// TwinCAT 3 PLC project TcoElements
// Title: TcoElements
// Company: Vortex.Library
// ProjectVersion: 0.6.0.913
// ProgramVersion: 3.1.4024.12
// libraries:
//   Tc2_Standard, * (Beckhoff Automation GmbH)
//   Tc2_System, * (Beckhoff Automation GmbH)
//   Tc3_Module, * (Beckhoff Automation GmbH)
//   TcoCore, 0.6.0.913 (Vortex.Library)
//   TcoUtilities, 0.6.0.913 (Vortex.Library)
// project tree:
//   Analog/TcoAi/ TcoAiAny.TcPOU, TcoAi.TcPOU, TcoAiConfig.TcDUT, TcoAiStatus.TcDUT
//   Analog/TcoAo/ TcoAoConfig.TcDUT, TcoAoStatus.TcDUT, TcoAo.TcPOU
//   Carousel/Base/ TcoCarouselBase.TcPOU
//   Carousel/Structs/ eTcoCarouselDirection.TcDUT, TcoCarouselConfig.TcDUT, TcoCarouselStatus.TcDUT
//   Carousel/Tasks/ TcoTurnTableTask.TcPOU
//   Carousel/ TcoCarousel.TcPOU
//   Digital/TcoDi/ TcoDi.TcPOU, TcoDiConfig.TcDUT
//   Digital/TcoDo/ TcoDo.TcPOU
//   / PlcTask.TcTTO
//   POUs/ MAIN.TcPOU
// real-time tasks:
//   TASK PlcTask: cycle T#10ms, priority 20, ADS port 350
//   TASK PlcTask1: cycle T#10ms, priority 21, ADS port 351

CONFIGURATION TcoElements
    RESOURCE PLC ON TwinCAT3
        TASK PlcTask(INTERVAL := T#10ms, PRIORITY := 20);
        PROGRAM MAIN WITH PlcTask : MAIN;
    END_RESOURCE
END_CONFIGURATION

// ---- Analog/TcoAo/TcoAoConfig.TcDUT
(*~
<docu>
    <summary>
        `TcoAo` settings/config structure.
    </summary>
</docu>
~*)
TYPE TcoAoConfig :
STRUCT
    (*~
        <docu>
            <summary>
                Lowest possible value of the raw input.
            </summary>
        </docu>
        ~*)
    RawLow : DINT;
    (*~
        <docu>
            <summary>
                Highest possible value of the raw input.
            </summary>
        </docu>
        ~*)
    RawHigh : DINT;
    (*~
        <docu>
            <summary>
                Lowest threshold of scaled value.
                `RealLow` and `RealHigh` should represent the real range of an continuous input.
            </summary>
        </docu>
        ~*)
    RealLow : REAL;
    (*~
        <docu>
            <summary>
                Highest threshold range of scaled value.
                `RealLow` and `RealHigh` should represent the real range of an continuous input.
            </summary>
        </docu>
        ~*)
    RealHigh : REAL;
    (*~
        <docu>
            <summary>
                Allows simple adjustment of the calculated value multiplying the value by factor of `Gain`.
            </summary>
        </docu>
        ~*)
    Gain : REAL := 1.0;
    (*~
        <docu>
            <summary>
                Allows simple adjustment of the calculated value by adding `Offset` value.
            </summary>
        </docu>
        ~*)
    Offset : REAL := 0.0;
END_STRUCT
END_TYPE

// ---- Analog/TcoAo/TcoAoStatus.TcDUT
(*~
<docu>
    <summary>
        `TcoAo` status structure.
    </summary>
</docu>
~*)
TYPE TcoAoStatus :
STRUCT
    (*~
        <docu>
            <summary>
                Absolute range of raw value.
            </summary>
        </docu>
        ~*)
    {attribute addProperty Name "<#Raw range#>"}
    RawRange : REAL;
    (*~
        <docu>
            <summary>
                Absolute range of real value.
            </summary>
        </docu>
        ~*)
    {attribute addProperty Name "<#Real range#>"}
    RealRange : REAL;
    (*~
        <docu>
            <summary>
                Current real value.
            </summary>
        </docu>
        ~*)
    {attribute addProperty Name "<#Unscaled value#>"}
    Unscaled : REAL;
END_STRUCT
END_TYPE

// ---- Carousel/Structs/eTcoCarouselDirection.TcDUT
TYPE eTcoCarouselDirection :
(
    Cw := 0,
    Ccw := 1
);
END_TYPE

// ---- Carousel/Structs/TcoCarouselConfig.TcDUT
(*~
<docu>
    <summary>
        `TcoCarousel` settings/config structure.
    </summary>
</docu>
~*)
TYPE TcoCarouselConfig :
STRUCT
    Direction : eTcoCarouselDirection;
    InfoTime : TIME := T#2S;
    ErrorTime : TIME := T#5S;
    NumberOfPositions : UINT;
    // Offset in respect to frist position.
    Offset : UINT;
END_STRUCT
END_TYPE

// ---- Carousel/Structs/TcoCarouselStatus.TcDUT
(*~
<docu>
    <summary>
        `TcCarousel` status structure.
    </summary>
</docu>
~*)
TYPE TcoCarouselStatus :
STRUCT
    ActionDescription : STRING(100);
    {attribute addProperty Name "<#In position#>"}
    InPosition : BOOL;
    {attribute addProperty Name "<#In precise position#>"}
    InPrecisePosition : BOOL;
    {attribute addProperty Name "<#Turn safety condition#>"}
    TurnSafetyCondition : BOOL;
    {attribute addProperty Name "<#Current position#>"}
    CurrentPosition : UINT;
    {attribute addProperty Name "<#Expected next position#>"}
    ExpectedNextPosition : UINT;
    {attribute addProperty Name "<#Positions#>" }
    Positions : ARRAY[0..20] OF UINT;
END_STRUCT
END_TYPE

// ---- Digital/TcoDi/TcoDiConfig.TcDUT
TYPE TcoDiConfig :
STRUCT
    IsFalseTimeOut : TIME := T#10S;
    IsTrueTimeOut : TIME := T#10S;
END_STRUCT
END_TYPE

// ---- Analog/TcoAi/TcoAiConfig.TcDUT
(*~
<docu>
    <summary>
        `TcoAi` settings/config structure.
    </summary>
</docu>
~*)
TYPE TcoAiConfig :
STRUCT
    (*~
        <docu>
            <summary>
                Lowest possible value of the raw input.
            </summary>
        </docu>
        ~*)
    RawLow : DINT;
    (*~
        <docu>
            <summary>
                Highest possible value of the raw input.
            </summary>
        </docu>
        ~*)
    RawHigh : DINT;
    (*~
        <docu>
            <summary>
                Lowest threshold of scaled value.
                `RealLow` and `RealHigh` should represent the real range of an continuous input.
            </summary>
        </docu>
        ~*)
    RealLow : REAL;
    (*~
        <docu>
            <summary>
                Highest threshold range of scaled value.
                `RealLow` and `RealHigh` should represent the real range of an continuous input.
            </summary>
        </docu>
        ~*)
    RealHigh : REAL;
    (*~
        <docu>
            <summary>
                Allows simple adjustment of the calculated value multiplying the value by factor of `Gain`.
            </summary>
        </docu>
        ~*)
    Gain : REAL := 1.0;
    (*~
        <docu>
            <summary>
                Allows simple adjustment of the calculated value by adding `Offset` value.
            </summary>
        </docu>
        ~*)
    Offset : REAL := 0.0;
END_STRUCT
END_TYPE

// ---- Analog/TcoAi/TcoAiStatus.TcDUT
(*~
<docu>
    <summary>
        `TcoAi` status structure.
    </summary>
</docu>
~*)
TYPE TcoAiStatus :
STRUCT
    (*~
        <docu>
            <summary>
                Absolute range of raw value.
            </summary>
        </docu>
        ~*)
    {attribute addProperty Name "<#Raw range#>"}
    RawRange : REAL;
    (*~
        <docu>
            <summary>
                Absolute range of real value.
            </summary>
        </docu>
        ~*)
    {attribute addProperty Name "<#Real range#>"}
    RealRange : REAL;
    (*~
        <docu>
            <summary>
                Current real value.
            </summary>
        </docu>
        ~*)
    {attribute addProperty Name "<#Scaled value#>"}
    Scaled : REAL;
END_STRUCT
END_TYPE

// ---- POUs/MAIN.TcPOU
PROGRAM INTERNAL MAIN

END_PROGRAM

// ---- Analog/TcoAi/TcoAiAny.TcPOU
(*~
    <docu>
        <summary>
                Generic component for monitoring of a continuous signal input. (e.g. AnalogSensor).
        </summary>
    </docu>
~*)
FUNCTION_BLOCK TcoAiAny EXTENDS TcoCore.TcoComponent
VAR_INPUT
    (*~
    <docu>
        <summary>
            Input  continious signal. Typically an `%I* : INT` or `%I* : DINT`  variable.
        </summary>
    </docu>
    ~*)
    inSignal : DINT;
    (*~
    <docu>
        <summary>
            Input additional symbol information about continious signal. Typically an `%I* : INT` or `%I* : DINT`  variable.
        </summary>
    </docu>
    ~*)
    inSignalInfo : TcoCore.TcoSignalInfo;
END_VAR
VAR
    (*~
    <docu>
        <summary>
            Backing variable for signal; this variable is used directly by the component. It updates `inoSingal` in FB body call.
        </summary>
    </docu>
    ~*)
    _signal : DINT;
END_VAR
VAR
    (*~
    <docu>
        <summary>
            Provides information about the input signal of this instance of `TcoAi`.
        </summary>
    </docu>
    ~*)
    {attribute addProperty Name "<#Signal#>"}
    _signalInfo : TcoCore.TcoSignalInfo;
    (*~
    <docu>
        <summary>
            Contains information about the settings and configuration of this instance of `TcoAi`.
        </summary>
    </docu>
    ~*)
    {attribute addProperty Name "<#Config#>"}
    _config : TcoAiConfig;
    (*~
    <docu>
        <summary>
            Contains information about the status if this instance of `TcoAi`.
        </summary>
    </docu>
    ~*)
    {attribute addProperty Name "<#Status#>"}
    _status : TcoAiStatus;
    _rawRange : REAL;
    _realRange : REAL;
    _scaled : REAL;
END_VAR

_signal := inSignal;
_signalInfo := inSignalInfo;
//------------------scale-------------------------
_rawRange := DINT_TO_REAL(_config.RawHigh - _config.RawLow);
_realRange := config.RealHigh - Config.RealLow;
_scaled := 0;

IF (_rawRange = 0) THEN
    Messenger.Warning('<#Division by zero: Verify values defined in config! (RawHigh,RawLow)#>');
    RETURN;
END_IF

IF (Config.Gain = 0) THEN
    Messenger.Warning('<#Invalid data: Gain is not defined!#>');
END_IF

_scaled := (DINT_TO_REAL(_signal - _config.RawLow)) / _rawRange;
_scaled := _scaled * _realRange;
_scaled := _scaled + _config.RealLow;
_scaled := _scaled * _config.Gain + _config.Offset;

//------------------------------------------------
IF (_scaled > _config.RealHigh) AND (_config.Gain <> 1 OR _config.Offset <> 0) THEN
    Messenger.Warning('<#Out of boundaries,check correction parameters (Gain,Ofset) in config!#>');
ELSIF (_scaled < _config.RealLow) AND (_config.Gain <> 1 OR _config.Offset <> 0) THEN
    Messenger.Warning('<#Out of boundaries,check correction parameters (Gain,Ofset) in config!#>');
END_IF

_status.RawRange := _rawRange;
_status.RealRange := _realRange;
_status.Scaled := _scaled;

PROPERTY Config : REFERENCE TO TcoAiConfig
GET
Config REF= _config;
END_GET
END_PROPERTY

{attribute 'hide'}
METHOD FB_init : BOOL
VAR_INPUT
    bInitRetains : BOOL; // if TRUE, the retain variables are initialized (warm start / cold start)
    bInCopyCode : BOOL; // if TRUE, the instance afterwards gets moved into the copy code (online change)
    ParentObject : ITcoObject;
END_VAR
END_METHOD

(*~
    <docu>
        <summary>
            Restores this instance to the Ready state. Can be called explicitly or from within one of the restore mechanisms.
        </summary>
    </docu>
~*)
METHOD Restore : ITcoRestorable
// No implementation needed for this componet.
END_METHOD

(*~
    <docu>
        <summary>
            Custom service (manual, maintenance) logic.
            This method must be implemented in derived class.
        </summary>
    </docu>
~*)
METHOD PROTECTED ServiceMode
END_METHOD

PROPERTY Status : REFERENCE TO TcoAiStatus
GET
Status REF= _status;
END_GET
END_PROPERTY

END_FUNCTION_BLOCK

// ---- Carousel/Base/TcoCarouselBase.TcPOU
FUNCTION_BLOCK ABSTRACT TcoCarouselBase EXTENDS TcoCore.TcoComponent
VAR_IN_OUT
    (*~
        <docu>
            <summary>
                In position sensor.
            </summary>
        </docu>
    ~*)
    inoInPosition : BOOL;
    (*~
        <docu>
            <summary>
                In precise position sensor.
            </summary>
        </docu>
    ~*)
    inoInPrecisePosition : BOOL;
END_VAR
VAR_IN_OUT
    (*~
        <docu>
            <summary>
                Enable turn signal.
            </summary>
        </docu>
    ~*)
    {attribute addProperty Name "<#Enable turn#>"}
    inoEnableTurn : BOOL;
    (*~
        <docu>
            <summary>
                Start turn  signal.
            </summary>
        </docu>
    ~*)
    {attribute addProperty Name "<#Start turn#>"}
    inoStartTurn : BOOL;
END_VAR
VAR
    {attribute addProperty Name "<#In position sensor#>"}
    _inPosition : BOOL;
    {attribute addProperty Name "<#In precise position sensor#>"}
    _inPrecisePosition : BOOL;
    (*~
        <docu>
            <summary>
                Enable turn  signal.
            </summary>
        </docu>
    ~*)
    {attribute addProperty Name "<#Enable turn table#>"}
    _enableTurn : BOOL;
    (*~
        <docu>
            <summary>
                Start trun signal.
            </summary>
        </docu>
    ~*)
    {attribute addProperty Name "<#Start turn table#>"}
    _startTurn : BOOL;
END_VAR
VAR
    {attribute addProperty Name "<#In position signal#>"}
    _InPositionSignalInfo : TcoCore.TcoSignalInfo;
    {attribute addProperty Name "<#In precise position signal#>"}
    _InPrecisePositionSignalInfo : TcoCore.TcoSignalInfo;
    {attribute addProperty Name "<#Enable turn signal#>"}
    _EnableTurnSignalInfo : TcoCore.TcoSignalInfo;
    {attribute addProperty Name "<#Start turn signal#>"}
    _StartTurnSignalInfo : TcoCore.TcoSignalInfo;
END_VAR

IF (__ISVALIDREF(inoInPosition)) THEN
    _inPosition := inoInPosition;
    _InPositionSignalInfo.GetSignalInfo(SIZEOF(inoInPosition), ADR(inoInPosition));
END_IF;

IF (__ISVALIDREF(inoInPrecisePosition)) THEN
    _inPrecisePosition := inoInPrecisePosition;
    _InPrecisePositionSignalInfo.GetSignalInfo(SIZEOF(inoInPrecisePosition), ADR(inoInPrecisePosition));
END_IF;

IF (__ISVALIDREF(inoEnableTurn)) THEN
    inoEnableTurn := _enableTurn;
    _EnableTurnSignalInfo.GetSignalInfo(SIZEOF(inoEnableTurn), ADR(inoEnableTurn));
END_IF;

IF (__ISVALIDREF(inoStartTurn)) THEN
    inoStartTurn := _startTurn;
    _StartTurnSignalInfo.GetSignalInfo(SIZEOF(inoStartTurn), ADR(inoStartTurn));
END_IF;

(*~
    <docu>
        <summary>
            Gets whether the carousel is in  position.
        </summary>
    </docu>
~*)
PROPERTY InPosition : bool
GET
InPosition := _inPosition;
END_GET
END_PROPERTY

(*~
    <docu>
        <summary>
            Gets whether the carousel is in precise position.
        </summary>
    </docu>
~*)
PROPERTY InPrecisePosition : bool
GET
InPrecisePosition := _inPrecisePosition;
END_GET
END_PROPERTY

(*~
    <docu>
        <summary>
            Restore all tasks of this instance into initial state.
        </summary>
    </docu>
~*)
METHOD Restore : ITcoRestorable
IF (TurnTask <> 0) THEN
    TurnTask.Restore();
END_IF;
END_METHOD

METHOD PROTECTED ServiceMode
END_METHOD

(*~
    <docu>
        <summary>
            Starts movement into work position.
        </summary>
    </docu>
~*)
METHOD Turn : TcoCore.ITcoTaskStatus
IF (TurnTask <> 0) THEN
    Turn := TurnTask.Invoke();
END_IF;
END_METHOD

(*~
    <docu>
        <summary>
            Gets the `TrunTask` task that controls the rotation from  position to next position in same direction.
            <remarks>
                <note type="important">
                    This is an abstract method and must be implemented in derived class.
                </note>
            </remarks>
        </summary>
    </docu>
~*)
PROPERTY PUBLIC ABSTRACT TurnTask : TcoCore.ITcoTask
GET
END_GET
END_PROPERTY

END_FUNCTION_BLOCK

// ---- Carousel/Tasks/TcoTurnTableTask.TcPOU
FUNCTION_BLOCK TcoTurnTableTask EXTENDS TcoCore.TcoTask
VAR_INPUT
    inSafetyCondition : BOOL;
END_VAR
VAR_IN_OUT
    inoInPosition : BOOL;
    inoInPrecisePosition : BOOL;
    inoEnableTurn : BOOL;
    inoStartTurn : BOOL;
    inoConfig : TcoCarouselConfig;
    inoStatus : TcoCarouselStatus;
END_VAR
VAR
    {attribute 'hide'}
    _progress : INT := 0;
    {attribute 'hide'}
    _infoTimer : TON;
    {attribute 'hide'}
    _errorTimer : TON;
    {attribute 'hide'}
    _varInfo : __SYSTEM.VAR_INFO;
    {attribute 'hide'}
    _sb : TcoCore.StringBuilder;
    _notInPositionMessage : TcoCore.TcoMessenger(THIS^);
END_VAR

IF (THIS^.Execute()) THEN
    IF _progress = 0 THEN
        IF NOT __ISVALIDREF(inoInPosition) THEN
            _varInfo := __VARINFO(inoInPosition);
            Messenger.Programming(_sb.Clear().Append('<#Invalid reference: #>').Append(_varInfo.Symbol).ToString()).Pin();
        ELSIF NOT __ISVALIDREF(inoInPrecisePosition) THEN
            _varInfo := __VARINFO(inoInPrecisePosition);
            Messenger.Programming(_sb.Clear().Append('<#Invalid reference: #>').Append(_varInfo.Symbol).ToString()).Pin();
        ELSIF NOT __ISVALIDREF(inoEnableTurn) THEN
            _varInfo := __VARINFO(inoEnableTurn);
            Messenger.Programming(_sb.Clear().Append('<#Invalid reference: #>').Append(_varInfo.Symbol).ToString()).Pin();
        ELSIF NOT __ISVALIDREF(inoStartTurn) THEN
            _varInfo := __VARINFO(inoStartTurn);
            Messenger.Programming(_sb.Clear().Append('<#Invalid reference: #>').Append(_varInfo.Symbol).ToString()).Pin();
        ELSIF NOT __ISVALIDREF(inoConfig) THEN
            _varInfo := __VARINFO(inoConfig);
            Messenger.Programming(_sb.Clear().Append('<#Invalid reference: #>').Append(_varInfo.Symbol).ToString()).Pin();
        ELSIF NOT __ISVALIDREF(inoStatus) THEN
            _varInfo := __VARINFO(inoStatus);
            Messenger.Programming(_sb.Clear().Append('<#Invalid reference: #>').Append(_varInfo.Symbol).ToString()).Pin();
        ELSE
            _progress := _progress + 1;
        END_IF
    END_IF

    IF _progress = 1 THEN
        _notInPositionMessage.OnCondition(NOT inoInPosition)
            .Error('<#Rotatiting started , but table is not in default position! Acknowledge this alarm if you still want to turn! #>').Pin();

        _progress := 10;
    END_IF;

    IF _progress = 10 THEN
        Messenger.Info('<#Calulate next expected Id position#>');

        IF inoStatus.CurrentPosition <> 0 THEN
            inoStatus.ExpectedNextPosition := GetIdentifierAtPosition(inoConfig.NumberOfPositions, inoStatus.Positions);
        END_IF;

        Messenger.OnCondition(inoStatus.CurrentPosition = 0 AND inoInPosition)
            .Error('<#Incorrectly coded current position. Check configuration of code bits! #>').Pin();

        IF inoStatus.CurrentPosition <> 0 AND inoInPosition THEN
            _progress := 20;
        ELSIF NOT _notInPositionMessage.Pinned THEN
            _progress := 20;
            _notInPositionMessage.UnPin();
        END_IF;
    END_IF;

    IF _progress = 20 THEN
        inoEnableTurn := TRUE;
        inoStartTurn := TRUE;
        Messenger.Info('<#Table turning. Trying to leave sensor#>');

        IF NOT inoInPosition THEN
            inoEnableTurn := FALSE;
            _progress := _progress + 10;
        END_IF
    END_IF;

    IF _progress = 30 THEN
        Messenger.Info('<#Table turning. Trying to reach sensor table in positon.#>');
        inoStartTurn := TRUE;

        IF inoInPosition THEN
            inoEnableTurn := FALSE;
            inoStartTurn := FALSE;
            _progress := _progress + 10;
        END_IF
    END_IF;

    IF _progress = 40 THEN
        Messenger
            .OnCondition(inoStatus.CurrentPosition > 0 AND_THEN inoStatus.ExpectedNextPosition <> GetIdentifierAtPosition(1, inoStatus.Positions))
            .Error(_sb.Clear()
                .Append('<#Table after turn does not have expected coding. Expected id at position #1 is#> ')
                .Append(UINT_TO_STRING(inoStatus.ExpectedNextPosition))
                .ToString()).Pin();

        IF (inoStatus.CurrentPosition > 0 AND inoStatus.ExpectedNextPosition = GetIdentifierAtPosition(1, inoStatus.Positions)) THEN
            THIS^.DoneWhen(TRUE);
        END_IF;
    END_IF;

    CallTimers(TRUE);
    THIS^.ThrowWhen(_errorTimer.Q);
END_IF

IF NOT inSafetyCondition THEN
    inoEnableTurn := FALSE;
    inoStartTurn := FALSE;
    Messenger.Error('<#Safety conditions to turn the table are not met.#>').Pin();
END_IF

METHOD CallTimers
VAR_INPUT
    inValue : BOOL;
END_VAR
IF __ISVALIDREF(inoConfig) THEN
    _infoTimer(IN := inValue, PT := THIS^.inoConfig.InfoTime);
    _errorTimer(IN := inValue, PT := THIS^.inoConfig.ErrorTime);
END_IF;
END_METHOD

{attribute 'hide'}
METHOD PUBLIC FB_init : BOOL
VAR_INPUT
    bInitRetains : BOOL; // if TRUE, the retain variables are initialized (warm start / cold start)
    bInCopyCode : BOOL; // if TRUE, the instance afterwards gets moved into the copy code (online change)
    ParentObject : ITcoObject;
END_VAR
END_METHOD

METHOD GetIdentifierAtPosition : UINT
VAR_INPUT
    inPosition : UINT;
    inPositions : ARRAY[0..20] OF UINT;
END_VAR
IF (inPosition < 1 OR inPosition > SIZEOF(inPositions)) THEN
    Messenger.Programming(Concat('<#Required position must be in range 1 - 20 but was:#>', UINT_TO_STRING(inPosition)));
    RETURN;
END_IF

GetIdentifierAtPosition := inPositions[inPosition - 1];
END_METHOD

(*~
    <docu>
        <summary>
            Executes when task is aborted.
        </summary>
    </docu>
~*)
METHOD PROTECTED OnAbort
IF __ISVALIDREF(inoStatus) THEN
    THIS^.inoStatus.ActionDescription := '<#Turning table was aborted, while not yet completed!#>';
END_IF;
END_METHOD

(*~
    <docu>
        <summary>
            Executes when task reaches the ```Done``` state .
        </summary>
    </docu>
~*)
METHOD PROTECTED OnDone
IF __ISVALIDREF(inoStatus) THEN
    THIS^.inoStatus.ActionDescription := '<#Truning table  was completed successfully.#>';
END_IF;
END_METHOD

METHOD PROTECTED OnError
IF __ISVALIDREF(inoStatus) THEN
    THIS^.inoStatus.ActionDescription := '<#Turning table finished with an error.#>';
END_IF;
END_METHOD

METHOD PROTECTED OnStart
IF __ISVALIDREF(inoStatus) THEN
    THIS^.inoStatus.ActionDescription := '<#Turning table started.#>';
END_IF;
END_METHOD

(*~
    <docu>
        <summary>
            Restores this instance to the Ready state. Can be called explicitly or from within one of the restore mechanisms.
            <para>
                See also <see cref="PlcDocu.TcoCore.TcoTask.AutoRestorable()"/>
            </para>
        </summary>
    </docu>
~*)
METHOD Restore : ITcoRestorable
SUPER^.Restore();
_progress := 0;
CallTimers(FALSE);
Messenger.UnPin();
_notInPositionMessage.UnPin();
END_METHOD

END_FUNCTION_BLOCK

// ---- Carousel/TcoCarousel.TcPOU
{attribute addProperty _turnTableName "<#Turn#>"}
{attribute addProperty _restoreName "<#Restore#>"}
FUNCTION_BLOCK TcoCarousel EXTENDS TcoCarouselBase
VAR_INPUT
    (*~
        <docu>
            <summary>
                This condition prevents the rotation of the table, possibly due to collisions with cylinders, axes, or other objects.
                Do not use signal from Light Curtain here.
            </summary>
        </docu>
    ~*)
    inSafetyCondition : BOOL;
    (*~
        <docu>
            <summary>
                The coded bites are stored in this word, which is valid for the base position of the carousel.
            </summary>
        </docu>
    ~*)
    inBasePositionNumber : WORD;
END_VAR
VAR
    {attribute addProperty Name "|[[1]Attribute_turnTableName]|"}
    _turnTask : TcoTurnTableTask(THIS^);
    {attribute addProperty Name "|[[1]Attribute_restoreName]|"}
    _restoreTask : TcoCore.TcoTask(THIS^);
    {attribute addProperty Name "<#Config#>"}
    _config : TcoCarouselConfig;
    {attribute addProperty Name "<#Status#>"}
    _status : TcoCarouselStatus;
END_VAR
VAR
    increment : INT;
    _index : INT;
    {attribute 'hide'}
    _positionsIdentifiersClear : ARRAY[0..20] OF UINT;
    _sb : TcoCore.StringBuilder;
    _basePositionNumber : WORD;
END_VAR

SUPER^(inoInPosition := inoInPosition,
    inoInPrecisePosition := inoInPrecisePosition,
    inoEnableTurn := inoEnableTurn,
    inoStartTurn := inoStartTurn);

_status.CurrentPosition := inBasePositionNumber;
_status.InPosition := _inPosition;
_status.InPrecisePosition := _inPrecisePosition;
_status.TurnSafetyCondition := inSafetyCondition;

IF (_config.NumberOfPositions <= 0) THEN
    Messenger.Programming('- <#Parameter number of positions is <= 0. The paremeters must be grater than 0.#>');
    RETURN;
END_IF

_status.Positions := _positionsIdentifiersClear;

IF (_config.OffSet = 0) THEN
    _config.OffSet := 1;
END_IF
// Calc position
_status.Positions[_config.NumberOfPositions - 1] := 1 + (1 - _config.Offset + _status.CurrentPosition) MOD _config.NumberOfPositions;

FOR _index := 1 TO UINT_TO_INT(_config.NumberOfPositions) - 1 DO
    _status.Positions[UINT_TO_INT(_config.NumberOfPositions) - 1 - _index] :=
        1 + ((_status.Positions[UINT_TO_INT(_config.NumberOfPositions) - _index]) MOD (_config.NumberOfPositions));
END_FOR
// Disables mutualy exclusive actions
_turnTask.Enabled := NOT _restoreTask.Busy;

_turnTask(inSafetyCondition := inSafetyCondition,
    inoInPosition := _inPosition,
    inoInPrecisePosition := _inPrecisePosition,
    inoEnableTurn := _enableTurn,
    inoStartTurn := _startTurn,
    inoConfig := _config,
    inoStatus := _status);

_restoreTask.Enabled := TRUE;

IF (_restoreTask.Execute()) THEN
    Restore();
    _restoreTask.DoneWhen(TRUE);
END_IF

// For further discussion about Status
IF (_turnTask.Busy) THEN
    _status.ActionDescription := 'Roatating table to next position ';
ELSIF (_restoreTask.Busy) THEN
    _status.ActionDescription := 'Restoring';
ELSE
    _status.ActionDescription := 'Idle';
END_IF

SUPER^(inoInPosition := inoInPosition,
    inoInPrecisePosition := inoInPrecisePosition,
    inoEnableTurn := inoEnableTurn,
    inoStartTurn := inoStartTurn);

(*~
    <docu>
        <summary>
            Aborts the turning when the condition is 'true'.
        </summary>
        <remarks>
                <note type="warning">
                    The call of this method will be effective only when called AFTER the initialization of the instance of given TcoCarousel.
                </note>
        </remarks>
    </docu>
~*)
METHOD Abort : BOOL
VAR_IN_OUT
    (*~
        <docu>
            <summary>
                Condition to abort the turning of the carousel.
            </summary>
        </docu>
    ~*)
    inoDisableCondition : BOOL;
END_VAR
VAR_INPUT
    (*~
        <docu>
            <summary>
                Condition to abort the movement of the carousel can be inverted by this parameter.
            </summary>
        </docu>
    ~*)
    Invert : BOOL;
END_VAR
VAR
    _signalInfo : TcoSignalInfo;
END_VAR
IF (_turnTask.Busy) AND inoDisableCondition AND NOT Invert THEN
    _signalInfo.GetSignalInfo(SIZEOF(inoDisableCondition), ADR(inoDisableCondition));
    Messenger.Build().Append('<#Turning table aborted due to#> : ').Append(_signalInfo.SymbolPath).As().AsError().Pin();
    _startTurn := FALSE;
    _enableTurn := FALSE;

    IF (__ISVALIDREF(THIS^.inoStartTurn)) THEN
        THIS^.inoStartTurn := FALSE;
    END_IF;

    IF (__ISVALIDREF(THIS^.inoEnableTurn)) THEN
        THIS^.inoEnableTurn := FALSE;
    END_IF;

    _turnTask.Abort();
ELSIF (_turnTask.Busy) AND inoDisableCondition AND Invert THEN
    _signalInfo.GetSignalInfo(SIZEOF(inoDisableCondition), ADR(inoDisableCondition));
    Messenger.Build().Append('<#Turning table aborted due to NOT #> : ').Append(_signalInfo.SymbolPath).As().AsError().Pin();
    _startTurn := FALSE;
    _enableTurn := FALSE;

    IF (__ISVALIDREF(THIS^.inoStartTurn)) THEN
        THIS^.inoStartTurn := FALSE;
    END_IF;

    IF (__ISVALIDREF(THIS^.inoEnableTurn)) THEN
        THIS^.inoEnableTurn := FALSE;
    END_IF;

    _turnTask.Abort();
END_IF
END_METHOD

(*~
    <docu>
        <summary>
            Gets the `StopTask` task that controls the stopping the turning carousel.
        </summary>
    </docu>
~*)
PROPERTY AbortTask : TcoCore.ITcoTask
GET
AbortTask := _restoreTask;
END_GET
END_PROPERTY

PROPERTY Config : REFERENCE TO TcoCarouselConfig
GET
Config REF= _config;
END_GET
END_PROPERTY

METHOD PUBLIC GetIdentifierAtPosition : UINT
VAR_INPUT
    inPosition : UINT;
END_VAR
GetIdentifierAtPosition := _turnTask.GetIdentifierAtPosition(inPosition := inPosition, inPositions := _status.Positions);
END_METHOD

(*~
    <docu>
        <summary>
            Restore all tasks of this instance into initial state.
        </summary>
    </docu>
~*)
METHOD Restore : ITcoRestorable
_turnTask.Restore();
_restoreTask.Abort();
_restoreTask.Restore();
_enableTurn := FALSE;
_startTurn := FALSE;
Messenger.UnPin();
END_METHOD

PROPERTY Status : REFERENCE TO TcoCarouselStatus
GET
Status REF= _status;
END_GET
END_PROPERTY

(*~
    <docu>
        <summary>
            Suspend the turning to next position when the condition is 'true'. Task is still bussy
        </summary>
        <remarks>
                <note type="warning">
                    The call of this method will be effective only when called AFTER the initialization of the instance of given TcoCarousel.
                </note>
        </remarks>
    </docu>
~*)
METHOD Suspend : BOOL
VAR_IN_OUT
    (*~
        <docu>
            <summary>
                Condition to suspend the movement of the carousel.
            </summary>
        </docu>
    ~*)
    inoDisableCondition : BOOL;
END_VAR
VAR_INPUT
    (*~
        <docu>
            <summary>
                Condition to suspend the movement of the carousel can be inverted by this parameter.
            </summary>
        </docu>
    ~*)
    Invert : BOOL;
END_VAR
VAR
    _signalInfo : TcoSignalInfo;
END_VAR
IF (_turnTask.Busy OR _startTurn OR _enableTurn) AND inoDisableCondition AND NOT Invert THEN
    _signalInfo.GetSignalInfo(SIZEOF(inoDisableCondition), ADR(inoDisableCondition));
    Messenger.Warning(_sb.Clear().Append('<#Turning table is suspended due to#> : ').Append(_signalInfo.SymbolPath).ToString());
    _startTurn := FALSE;
    _enableTurn := FALSE;

    IF (__ISVALIDREF(THIS^.inoStartTurn)) THEN
        THIS^.inoStartTurn := FALSE;
    END_IF;

    IF (__ISVALIDREF(THIS^.inoEnableTurn)) THEN
        THIS^.inoEnableTurn := FALSE;
    END_IF;
ELSIF (_turnTask.Busy OR _startTurn OR _enableTurn) AND inoDisableCondition AND Invert THEN
    _signalInfo.GetSignalInfo(SIZEOF(inoDisableCondition), ADR(inoDisableCondition));
    Messenger.Warning(_sb.Clear().Append('<#Turning table is suspended due to NOT #> : ').Append(_signalInfo.SymbolPath).ToString());
    _startTurn := FALSE;
    _enableTurn := FALSE;

    IF (__ISVALIDREF(THIS^.inoStartTurn)) THEN
        THIS^.inoStartTurn := FALSE;
    END_IF;

    IF (__ISVALIDREF(THIS^.inoEnableTurn)) THEN
        THIS^.inoEnableTurn := FALSE;
    END_IF;
END_IF
END_METHOD

METHOD SuspendExpression : BOOL
VAR_INPUT
    inDisableCondition : BOOL;
    inMessage : STRING;
END_VAR
IF (_turnTask.Busy OR _startTurn OR _enableTurn) AND inDisableCondition THEN
    Messenger.Warning(CONCAT('<#Rotating is suspended due to#> : ', inMessage));
    _startTurn := FALSE;
    _enableTurn := FALSE;

    IF (__ISVALIDREF(THIS^.inoStartTurn)) THEN
        THIS^.inoStartTurn := FALSE;
    END_IF;

    IF (__ISVALIDREF(THIS^.inoEnableTurn)) THEN
        THIS^.inoEnableTurn := FALSE;
    END_IF;
END_IF;
END_METHOD

(*~
    <docu>
        <summary>
            Gets the `TurnTask` task that controls the moving of the carousel to next position.
        </summary>
    </docu>
~*)
PROPERTY TurnTask : TcoCore.ITcoTask
GET
TurnTask := _turnTask;
END_GET
END_PROPERTY

END_FUNCTION_BLOCK

// ---- Digital/TcoDi/TcoDi.TcPOU
(*~
    <docu>
        <summary>
                Generic component for monitoring of an input. (e.g. DigitalSensor).
        </summary>
    </docu>
~*)
FUNCTION_BLOCK TcoDi EXTENDS TcoCore.TcoComponent
VAR_IN_OUT
    (*~
    <docu>
        <summary>
            Input signal. Typically an `%I*` variable.
        </summary>
    </docu>
    ~*)
    inoSignal : BOOL;
END_VAR
VAR
    (*~
    <docu>
        <summary>
            Backing variable for signal; this variable is used directly by the component. It updates `inoSingal` in FB body call.
        </summary>
    </docu>
    ~*)
    _signal : BOOL;
END_VAR
VAR
    {attribute addProperty Name "<#Signal#>"}
    _signalInfo : TcoCore.TcoSignalInfo;
    {attribute addProperty Name "<#Check On#>"}
    {attribute addProperty ToolTip "<#Checks that the input is on#>"}
    _isTrueTask : TcoCore.TcoTask(THIS^);
    {attribute addProperty ToolTip "<#Checks that the input is off#>"}
    {attribute addProperty Name "<#Check Off#>"}
    _isFalseTask : TcoCore.TcoTask(THIS^);
    _config : TcoDiConfig;
    _isFalseTimeOutTimers : Tc2_Standard.TON;
    _isTrueTimeOutTimers : Tc2_Standard.TON;
END_VAR

IF (__ISVALIDREF(inoSignal)) THEN
    _signalInfo.GetSignalInfo(SIZEOF(inoSignal), ADR(inoSignal));
    _signal := inoSignal;
END_IF;

IF (_isTrueTask.Execute()) THEN
    _isTrueTask.DoneWhen(IsTrue);
END_IF

IF (_isFalseTask.Execute()) THEN
    _isFalseTask.DoneWhen(IsFalse);
END_IF

PROPERTY Config : REFERENCE TO TcoDiConfig
GET
Config REF= _config;
END_GET
END_PROPERTY

METHOD FB_init : BOOL
VAR_INPUT
    bInitRetains : BOOL; // if TRUE, the retain variables are initialized (warm start / cold start)
    bInCopyCode : BOOL; // if TRUE, the instance afterwards gets moved into the copy code (online change)
    ParentObject : ITcoObject;
END_VAR
END_METHOD

(*~
    <docu>
        <summary>
            Gets 'true' when monitor signal is 'off/false/logical 0'.
            Generates message when the returning 'false'.
        </summary>
    </docu>
~*)
{attribute 'monitoring' := 'variable'}
PROPERTY IsFalse : BOOL
GET
IsFalse := NOT _signal;
_isFalseTimeOutTimers(IN := NOT IsFalse, PT := _config.IsFalseTimeOut);

IF (NOT IsFalse) THEN
    Messenger.Info('<#Expecting `negative` signal#>');
END_IF;

IF (_isFalseTimeOutTimers.Q) THEN
    Messenger.Warning('<#Expecting `negative` signal#>');
END_IF;
END_GET
END_PROPERTY

(*~
    <docu>
        <summary>
            Gets 'true' when monitor signal is 'on/true/logical 1'.
            Generates message when the returning 'false'.
        </summary>
    </docu>
~*)
{attribute 'monitoring' := 'variable'}
PROPERTY IsTrue : BOOL
GET
IsTrue := _signal;
_isTrueTimeOutTimers(IN := NOT IsTrue, PT := _config.IsFalseTimeOut);

IF (NOT IsTrue) THEN
    Messenger.Info('<#Expecting `positive` signal#>');
END_IF;

IF (_isTrueTimeOutTimers.Q) THEN
    Messenger.Warning('<#Expecting `positive` signal#>');
END_IF;
END_GET
END_PROPERTY

(*~
    <docu>
        <summary>
            Restores this instance to the Ready state. Can be called explicitly or from within one of the restore mechanisms.
        </summary>
    </docu>
~*)
METHOD Restore : ITcoRestorable
// No implementation needed for this componet.
END_METHOD

(*~
    <docu>
        <summary>
            Custom service (manual, maintenance) logic.
            This method must be implemented in derived class.
        </summary>
    </docu>
~*)
METHOD PROTECTED ServiceMode
END_METHOD

PROPERTY PUBLIC Signal : Bool
GET
Signal := _signal;
END_GET
END_PROPERTY

END_FUNCTION_BLOCK

// ---- Digital/TcoDo/TcoDo.TcPOU
(*~
    <docu>
        <summary>
                Generic component for discrete control of an output.
        </summary>
    </docu>
~*)
FUNCTION_BLOCK TcoDo EXTENDS TcoCore.TcoComponent
VAR_IN_OUT
    (*~
    <docu>
        <summary>
            Controlled signal. Typically an `%Q*` variable.
        </summary>
    </docu>
    ~*)
    inoSignal : BOOL;
END_VAR
VAR
    (*~
    <docu>
        <summary>
            Backing variable for signal; this variable is used directly by the component. It updates `inoSingal` in FB body call.
        </summary>
    </docu>
    ~*)
    _signal : BOOL;
END_VAR
VAR
    {attribute addProperty Name "<#Signal#>"}
    _signalInfo : TcoCore.TcoSignalInfo;
    {attribute addProperty Name "<#On#>"}
    {attribute addProperty ToolTip "<#Sets the output#>"}
    _setTask : TcoCore.TcoTask(THIS^);
    {attribute addProperty ToolTip "<#Resets the output#>"}
    {attribute addProperty Name "<#Off#>"}
    _resetTask : TcoCore.TcoTask(THIS^);
END_VAR

IF (__ISVALIDREF(inoSignal)) THEN
    _signalInfo.GetSignalInfo(SIZEOF(inoSignal), ADR(inoSignal));
    inoSignal := _signal;
END_IF;

IF (_setTask.Execute()) THEN
    _setTask.DoneWhen(Set());
END_IF

IF (_resetTask.Execute()) THEN
    _resetTask.DoneWhen(Reset());
END_IF

METHOD FB_init : BOOL
VAR_INPUT
    bInitRetains : BOOL; // if TRUE, the retain variables are initialized (warm start / cold start)
    bInCopyCode : BOOL; // if TRUE, the instance afterwards gets moved into the copy code (online change)
    ParentObject : ITcoObject;
END_VAR
END_METHOD

(*~
    <docu>
        <summary>
            Gets 'true' when monitor signal is 'off/false/logical 0'.
            Generates message when the returning 'false'.
        </summary>
    </docu>
~*)
{attribute 'monitoring' := 'variable'}
PROPERTY IsFalse : BOOL
GET
IsFalse := NOT _signal;

IF (NOT IsFalse) THEN
    Messenger.Info('<#Expecting `negative` signal#>');
END_IF;
END_GET
END_PROPERTY

(*~
    <docu>
        <summary>
            Gets 'true' when monitor signal is 'on/true/logical 1'.
            Generates message when the returning 'false'.
        </summary>
    </docu>
~*)
{attribute 'monitoring' := 'variable'}
PROPERTY IsTrue : BOOL
GET
IsTrue := _signal;

IF (NOT IsTrue) THEN
    Messenger.Info('<#Expecting `positive` signal#>');
END_IF;
END_GET
END_PROPERTY

(*~
    <docu>
        <summary>
            Sets controlled signal into 'off/false/logical 0'.
        </summary>
    </docu>
~*)
METHOD Reset : BOOL
Messenger.Trace('<#Reseting signal (off/false)#>');
_signal := FALSE;
Reset := TRUE;
END_METHOD

(*~
    <docu>
        <summary>
            Restores this instance to the Ready state. Can be called explicitly or from within one of the restore mechanisms.
        </summary>
    </docu>
~*)
METHOD Restore : ITcoRestorable
// No implementation needed for this componet.
END_METHOD

(*~
    <docu>
        <summary>
            Custom service (manual, maintenance) logic.
            This method must be implemented in derived class.
        </summary>
    </docu>
~*)
METHOD PROTECTED ServiceMode
END_METHOD

(*~
    <docu>
        <summary>
            Sets controlled signal into 'on/true/logical 1'.
        </summary>
    </docu>
~*)
METHOD PUBLIC Set : BOOL
Messenger.Trace('<#Setting signal (on/true)#>');
_signal := TRUE;
Set := TRUE;
END_METHOD

PROPERTY PUBLIC Signal : Bool
GET
Signal := _signal;
END_GET
END_PROPERTY

END_FUNCTION_BLOCK

// ---- Analog/TcoAi/TcoAi.TcPOU
(*~
    <docu>
        <summary>
                Generic component for monitoring of a continuous signal input. (e.g. AnalogSensor).
        </summary>
    </docu>
~*)
FUNCTION_BLOCK TcoAi EXTENDS TcoCore.TcoComponent
VAR_IN_OUT
    (*~
    <docu>
        <summary>
            Input  continious signal. Typically an `%I* : INT` or `%I* : DINT`  variable.
        </summary>
    </docu>
    ~*)
    inoSignal : DINT;
END_VAR
VAR
    (*~
    <docu>
        <summary>
            Backing variable for signal; this variable is used directly by the component. It updates `inoSingal` in FB body call.
        </summary>
    </docu>
    ~*)
    _signal : DINT;
END_VAR
VAR
    (*~
    <docu>
        <summary>
            Provides information about the input signal of this instance of `TcoAi`.
        </summary>
    </docu>
    ~*)
    {attribute addProperty Name "<#Signal#>"}
    _signalInfo : TcoCore.TcoSignalInfo;
    (*~
    <docu>
        <summary>
            Contains information about the settings and configuration of this instance of `TcoAi`.
        </summary>
    </docu>
    ~*)
    {attribute addProperty Name "<#Config#>"}
    _config : TcoAiConfig;
    (*~
    <docu>
        <summary>
            Contains information about the status if this instance of `TcoAi`.
        </summary>
    </docu>
    ~*)
    {attribute addProperty Name "<#Status#>"}
    _status : TcoAiStatus;
    _rawRange : REAL;
    _realRange : REAL;
    _scaled : REAL;
END_VAR

IF (__ISVALIDREF(inoSignal)) THEN
    _signalInfo.GetSignalInfo(SIZEOF(inoSignal), ADR(inoSignal));
    _signal := inoSignal;
END_IF;
//------------------scale-------------------------
_rawRange := DINT_TO_REAL(_config.RawHigh - _config.RawLow);
_realRange := config.RealHigh - Config.RealLow;
_scaled := 0;

IF (_rawRange = 0) THEN
    Messenger.Warning('<#Division by zero: Verify values defined in config! (RawHigh,RawLow)#>');
    RETURN;
END_IF

IF (Config.Gain = 0) THEN
    Messenger.Warning('<#Invalid data: Gain is not defined!#>');
END_IF

_scaled := (DINT_TO_REAL(_signal - _config.RawLow)) / _rawRange;
_scaled := _scaled * _realRange;
_scaled := _scaled + _config.RealLow;
_scaled := _scaled * _config.Gain + _config.Offset;

//------------------------------------------------
IF (_scaled > _config.RealHigh) AND (_config.Gain <> 1 OR _config.Offset <> 0) THEN
    Messenger.Warning('<#Out of boundaries,check correction parameters (Gain,Ofset) in config!#>');
ELSIF (_scaled < _config.RealLow) AND (_config.Gain <> 1 OR _config.Offset <> 0) THEN
    Messenger.Warning('<#Out of boundaries,check correction parameters (Gain,Ofset) in config!#>');
END_IF

_status.RawRange := _rawRange;
_status.RealRange := _realRange;
_status.Scaled := _scaled;

PROPERTY Config : REFERENCE TO TcoAiConfig
GET
Config REF= _config;
END_GET
END_PROPERTY

{attribute 'hide'}
METHOD FB_init : BOOL
VAR_INPUT
    bInitRetains : BOOL; // if TRUE, the retain variables are initialized (warm start / cold start)
    bInCopyCode : BOOL; // if TRUE, the instance afterwards gets moved into the copy code (online change)
    ParentObject : ITcoObject;
END_VAR
END_METHOD

(*~
    <docu>
        <summary>
            Restores this instance to the Ready state. Can be called explicitly or from within one of the restore mechanisms.
        </summary>
    </docu>
~*)
METHOD Restore : ITcoRestorable
// No implementation needed for this componet.
END_METHOD

(*~
    <docu>
        <summary>
            Custom service (manual, maintenance) logic.
            This method must be implemented in derived class.
        </summary>
    </docu>
~*)
METHOD PROTECTED ServiceMode
END_METHOD

PROPERTY Status : REFERENCE TO TcoAiStatus
GET
Status REF= _status;
END_GET
END_PROPERTY

END_FUNCTION_BLOCK

// ---- Analog/TcoAo/TcoAo.TcPOU
(*~
    <docu>
        <summary>
                Generic component for continious control of an output.(e. g. Continious analog sensor)
        </summary>
    </docu>
~*)
FUNCTION_BLOCK TcoAo EXTENDS TcoCore.TcoComponent
VAR_IN_OUT
    (*~
    <docu>
        <summary>
            Controlled signal. Typically an `%Q* : INT` ,`%Q* : DINT` variable.
        </summary>
    </docu>
    ~*)
    inoSignal : DINT;
END_VAR
VAR
    (*~
    <docu>
        <summary>
            Backing variable for signal; this variable is used directly by the component. It updates `inoSingal` in FB body call.
        </summary>
    </docu>
    ~*)
    _signal : DINT;
END_VAR
VAR
    {attribute addProperty Name "<#Signal#>"}
    _signalInfo : TcoCore.TcoSignalInfo;
    {attribute addProperty Name "<#Config#>"}
    _config : TcoAoConfig;
    {attribute addProperty Name "<#Status#>"}
    _status : TcoAoStatus;
    {attribute addProperty Name "<#Setpoint#>"}
    _requiredValue : REAL;
    _rawRange : REAL;
    _realRange : REAL;
    _unscaled : REAL;
END_VAR

IF (__ISVALIDREF(inoSignal)) THEN
    _signalInfo.GetSignalInfo(SIZEOF(inoSignal), ADR(inoSignal));
    inoSignal := _signal;
END_IF;
//------------------unscale-------------------------
_rawRange := DINT_TO_REAL(_config.RawHigh - _config.RawLow);
_realRange := config.RealHigh - Config.RealLow;
_unscaled := 0;

IF (_rawRange = 0) THEN
    Messenger.Error('<#Division by zero: Verify values defined in config! (RawHigh,RawLow)#>');
    RETURN;
END_IF

IF (Config.Gain = 0) THEN
    Messenger.Warning('<#Invalid data: Gain is not defined!#>');
END_IF

_unscaled := (_requiredValue - _config.RealLow) / _realRange;
_unscaled := _unscaled * _rawRange;
_unscaled := _unscaled + DINT_TO_REAL(_config.RawLow);
_unscaled := _unscaled * _config.Gain + _config.Offset;

//------------------------------------------------
IF (_unscaled > DINT_TO_REAL(_config.RawHigh)) AND (_config.Gain <> 1 OR _config.Offset <> 0) THEN
    Messenger.Warning('<#Out of boundaries,check correction parameters (Gain,Ofset) in config!#>');
ELSIF (_unscaled < DINT_TO_REAL(_config.RawLow)) AND (_config.Gain <> 1 OR _config.Offset <> 0) THEN
    Messenger.Warning('<#Out of boundaries,check correction parameters (Gain,Ofset) in config!#>');
END_IF

_signal := REAL_TO_DINT(_unscaled);
_status.RawRange := _rawRange;
_status.RealRange := _realRange;
_status.Unscaled := _unscaled;

IF (__ISVALIDREF(inoSignal)) THEN
    inoSignal := _signal;
END_IF;

PROPERTY Config : REFERENCE TO TcoAoConfig
GET
Config REF= _config;
END_GET
END_PROPERTY

{attribute 'hide'}
METHOD FB_init : BOOL
VAR_INPUT
    bInitRetains : BOOL; // if TRUE, the retain variables are initialized (warm start / cold start)
    bInCopyCode : BOOL; // if TRUE, the instance afterwards gets moved into the copy code (online change)
    ParentObject : ITcoObject;
END_VAR
END_METHOD

PROPERTY PUBLIC RequiredValue : REAL
GET
RequiredValue := _requiredValue;
END_GET
SET
_requiredValue := RequiredValue;
END_SET
END_PROPERTY

(*~
    <docu>
        <summary>
            Restores this instance to the Ready state. Can be called explicitly or from within one of the restore mechanisms.
        </summary>
    </docu>
~*)
METHOD Restore : ITcoRestorable
// No implementation needed for this componet.
END_METHOD

(*~
    <docu>
        <summary>
            Custom service (manual, maintenance) logic.
            This method must be implemented in derived class.
        </summary>
    </docu>
~*)
METHOD PROTECTED ServiceMode
END_METHOD

PROPERTY Status : REFERENCE TO TcoAoStatus
GET
Status REF= _status;
END_GET
END_PROPERTY

END_FUNCTION_BLOCK
